// This function has been automatically generated from the project information.
{attribute 'signature_flag' := '1073741824'}
{attribute 'TcGenerated'}
{attribute 'no-analysis'}
FUNCTION F_GetTitle : WSTRING
VAR_INPUT
	
END_VAR

F_GetTitle := "Tc3_CRC";

END_FUNCTION

(* stored: Version 1.1.0.1
   POU F_GetTitle: Id {98c97911-b0f5-4717-8ac5-9b1014dfd600}, SpecialFunc None *)
